{attribute 'GeneratedUsingTerminal: EK1100-0000-0018'}
{attribute addProperty BoxType "EK1100-0000-0018"}
{attribute addProperty Id "TcTerminals210_1BK1250TcTerminals210_1BK1250_A7ABB5AA0"}
{attribute addProperty CRC "1551336313"}
{attribute addProperty Size "0"}
TYPE TcTerminals210_EK1100_1_5C778379 EXTENDS EK1100_AB5A9467 :
STRUCT
	{attribute addProperty Name "TcTerminals210_1BK1250"}
	{attribute addProperty PreviousPort "TcTerminals210_EK1100_1 : B"}
	TcTerminals210_1BK1250 : TcTerminals210_1BK1250_A7ABB5AA;
END_STRUCT
END_TYPE

(* stored: Version 1.2.0.0, ProductVersion 3.1.4024.9
   DUT TcTerminals210_EK1100_1_5C778379: Id {c9a45ba8-4f2c-4941-8d12-28b4b9e9569b} *)
